PROGRAM TEST
VAR
END_VAR

END_PROGRAM

(* stored: Version 1.1.0.1, ProductVersion 3.1.4024.12
   POU TEST: Id {c9f63f39-ca52-4283-840c-538bd597e0b6}, SpecialFunc None *)
